// SIMATIC STEP 7 (V5.x) project GYDS2018
// CPU: CPU 315-2 PN/DP
// station: 硬件
// station: SIMATIC 300(1)
// station: P_ADR_BUS
// program: S7 程序(2)

SYMBOL_TABLE
"VAT_1"	VAT 1	
END_SYMBOL_TABLE

FUNCTION FC 1 : VOID
VERSION : 0.1
VAR_INPUT
  IN0 : INT ;
END_VAR
VAR_OUTPUT
  OUT1 : REAL ;
END_VAR
VAR_TEMP
  TEMP2 : INT ;
  TEMP3 : DINT ;
  TEMP4 : REAL ;
END_VAR
BEGIN
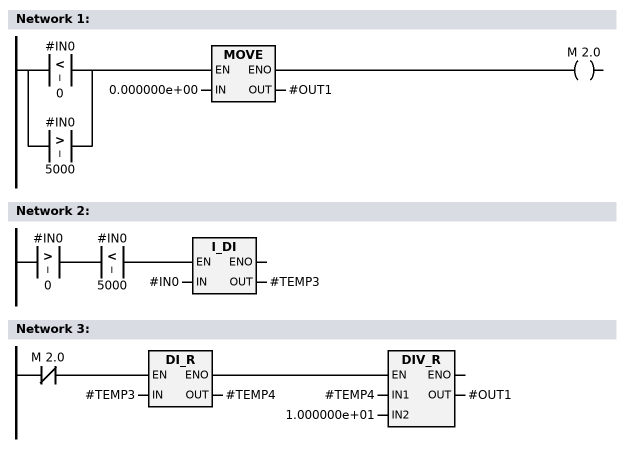
NETWORK
TITLE =
      A(;
      O(;
      L     #IN0;
      L     0;
      <I;
      );
      O(;
      L     #IN0;
      L     5000;
      >I;
      );
      );
      JNB   _001;
      L     0.000000e+00;
      T     #OUT1;
      SET;
      SAVE;
      CLR;
_001: A     BR;
      =     M 2.0;
NETWORK
TITLE =
      A(;
      L     #IN0;
      L     0;
      >I;
      );
      A(;
      L     #IN0;
      L     5000;
      <I;
      );
      JNB   _002;
      L     #IN0;
      ITD;
      T     #TEMP3;
_002: NOP   0;
NETWORK
TITLE =
      A(;
      AN    M 2.0;
      JNB   _003;
      L     #TEMP3;
      DTR;
      T     #TEMP4;
      SET;
      SAVE;
      CLR;
_003: A     BR;
      );
      JNB   _004;
      L     #TEMP4;
      L     1.000000e+01;
      /R;
      T     #OUT1;
_004: NOP   0;
END_FUNCTION

FUNCTION FC 16 : VOID
AUTHOR : LI_CS
VERSION : 0.1
BEGIN
// (block stored without names or comments; labels and parameter names are numbered)
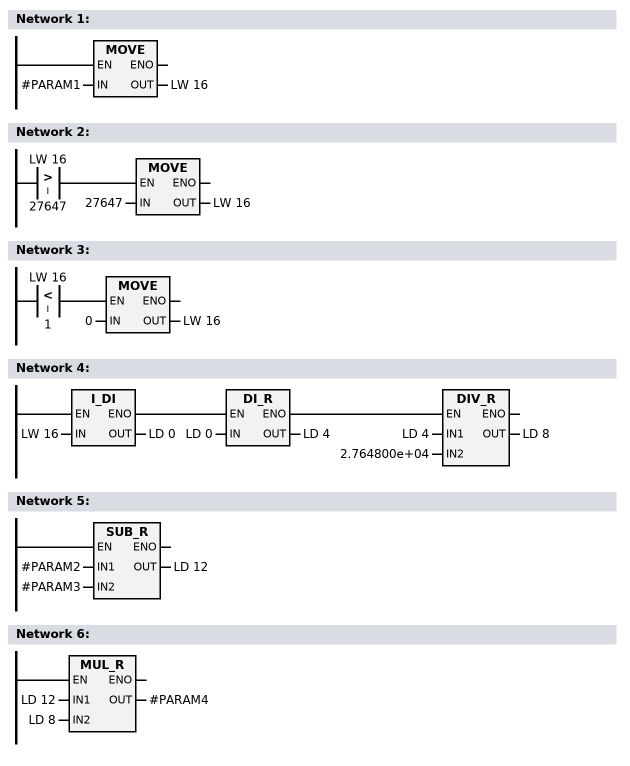
NETWORK
TITLE =
      L     #PARAM1;
      T     LW 16;
      NOP   0;
NETWORK
TITLE =
      A(;
      L     LW 16;
      L     27647;
      >I;
      );
      JNB   M001;
      L     27647;
      T     LW 16;
M001: NOP   0;
NETWORK
TITLE =
      A(;
      L     LW 16;
      L     1;
      <I;
      );
      JNB   M002;
      L     0;
      T     LW 16;
M002: NOP   0;
NETWORK
TITLE =
      A(;
      A(;
      L     LW 16;
      ITD;
      T     LD 0;
      SET;
      SAVE;
      CLR;
      A     BR;
      );
      JNB   M003;
      L     LD 0;
      DTR;
      T     LD 4;
      SET;
      SAVE;
      CLR;
M003: A     BR;
      );
      JNB   M004;
      L     LD 4;
      L     2.764800e+04;
      /R;
      T     LD 8;
M004: NOP   0;
NETWORK
TITLE =
      L     #PARAM2;
      L     #PARAM3;
      -R;
      T     LD 12;
      NOP   0;
NETWORK
TITLE =
      L     LD 12;
      L     LD 8;
      *R;
      T     #PARAM4;
      NOP   0;
END_FUNCTION

DATA_BLOCK DB 1
VERSION : 0.1
  STRUCT
   TEMP_TAG1 : REAL ;	//TEMP_TAG1
  END_STRUCT ;	
BEGIN
END_DATA_BLOCK

ORGANIZATION_BLOCK OB 1
TITLE = "Main Program Sweep (Cycle)"
VERSION : 0.1
VAR_TEMP
  OB1_EV_CLASS : BYTE ;	//Bits 0-3 = 1 (Coming event), Bits 4-7 = 1 (Event class 1)
  OB1_SCAN_1 : BYTE ;	//1 (Cold restart scan 1 of OB 1), 3 (Scan 2-n of OB 1)
  OB1_PRIORITY : BYTE ;	//Priority of OB Execution
  OB1_OB_NUMBR : BYTE ;	//1 (Organization block 1, OB1)
  OB1_RESERVED_1 : BYTE ;	//Reserved for system
  OB1_RESERVED_2 : BYTE ;	//Reserved for system
  OB1_PREV_CYCLE : INT ;	//Cycle time of previous OB1 scan (milliseconds)
  OB1_MIN_CYCLE : INT ;	//Minimum cycle time of OB1 (milliseconds)
  OB1_MAX_CYCLE : INT ;	//Maximum cycle time of OB1 (milliseconds)
  OB1_DATE_TIME : DATE_AND_TIME ;	//Date and time OB1 started
END_VAR
BEGIN
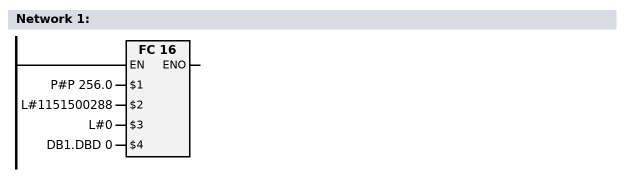
NETWORK
TITLE =
      CALL  FC 16 (
           $1                       := P#P 256.0,
           $2                       := L#1151500288,
           $3                       := L#0,
           $4                       := DB1.DBD 0);
      NOP   0;
END_ORGANIZATION_BLOCK
